# B&R Automation Studio project Lab1
Automation Studio 4.5.2.102

## Configuration Config1

### Hardware
```
4PP065_0351_P74 : 4PP065.0351-P74 v1.0.4.0
  Connector IF5:
    ActivateDevice = 1
  ConfigurationID = lab1_Config1
  KeyMappingFile = VC\4PP065_0351_P74.dis
```

## Logical view

### Program Logical/Program1

#### Variables.var
```iecst
VAR
	enable : BOOL := TRUE;
	counter : REAL := 0;
	speed : REAL := 0;
	fb_motor : FB_Motor;
	fb_motor2 : FB_Motor;
	fb_regulator : FB_Regulator;
END_VAR
```

#### Cyclic.c
```c
#include <bur/plctypes.h>

#ifdef _DEFAULT_INCLUDES
	#include <AsDefault.h>
#endif

void _CYCLIC ProgramCyclic(void)
{
	if (enable)
	{
		if (counter == 200)
		{
			speed = 0;
		}
		else if (counter == 50)
		{
			speed = 50;
		}
		if (counter < 201)
			counter++;

		fb_regulator.e = speed-fb_motor.w;
		FB_Regulator(&fb_regulator);
		fb_motor.u = fb_regulator.u;
		fb_motor2.u = speed * fb_motor2.ke;
		FB_Motor(&fb_motor);
		FB_Motor(&fb_motor2);
	}
}
```

#### Init.c
```c
#include <bur/plctypes.h>

#ifdef _DEFAULT_INCLUDES
	#include <AsDefault.h>
#endif

void _INIT ProgramInit(void)
{
	fb_motor.dt = 0.01;
	fb_motor.ke = 7.2;
	fb_motor.Tm = 0.1;
	fb_motor.u = 0;
	fb_motor.phi = 0;
	fb_motor.integrator1.dt = 0.01 / fb_motor.Tm;
	fb_motor.integrator2.dt = 0.01;

	fb_motor2.dt = 0.01;
	fb_motor2.ke = 7.2;
	fb_motor2.Tm = 0.1;
	fb_motor2.u = 0;
	fb_motor2.phi = 0;
	fb_motor2.integrator1.dt = 0.01  / fb_motor2.Tm;
	fb_motor2.integrator2.dt = 0.01;

	fb_regulator.dt = 0.01;
	fb_regulator.integrator.dt = 0.01;
	fb_regulator.k_i = 7.2;
	fb_regulator.k_p = 0.24 * 3;
	fb_regulator.max_abs_value = 24.0;

	speed = 0;
	counter = 0;
}
```
